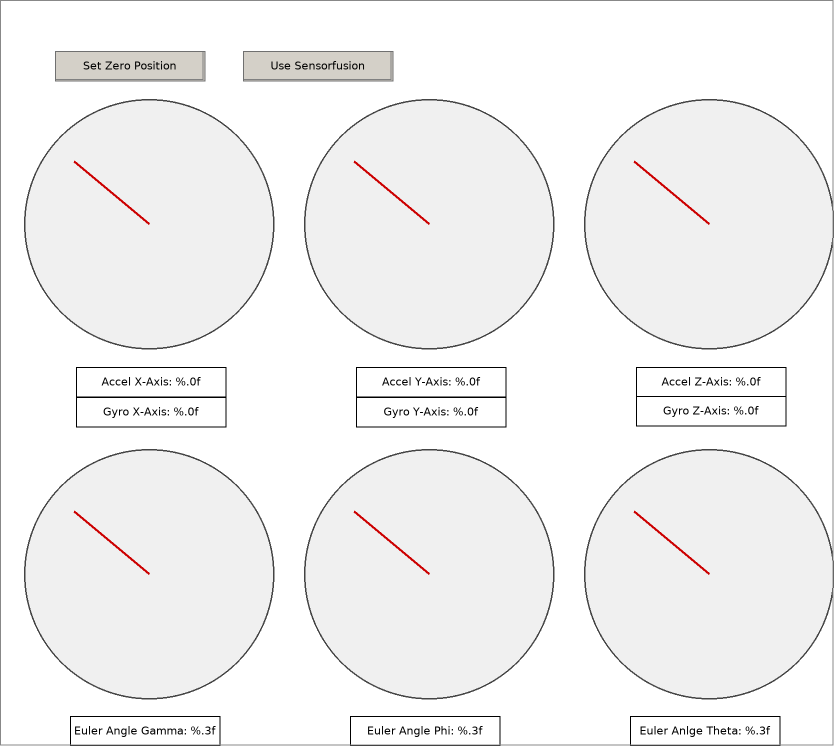
VISUALIZATION Visualization  // 834x746
    Meter360 (24,99 250x250), value: MAIN.AccAxis[0], style: Meter-Meter360-Gray, scale format: %d, scale -2000..2000
        p518627256: °
    Rectangle (76,367 150x30), "Accel X-Axis: %.0f", text variable: MAIN.AccAxis[0]
    Button (55,51 150x30), "Set Zero Position", colour toggle: MAIN.bReady
        p2175578022: 16#FF808080
        p573394764: 16#FF80FF80
        tap MAIN.bReset
    Meter360 (304,99 250x250), value: MAIN.AccAxis[1], style: Meter-Meter360-Gray, scale format: %d, scale -2000..2000
        p518627256: °
    Rectangle (356,367 150x30), "Accel Y-Axis: %.0f", text variable: MAIN.AccAxis[1]
    Meter360 (584,99 250x250), value: MAIN.AccAxis[2], style: Meter-Meter360-Gray, scale format: %d, scale -2000..2000
        p518627256: °
    Rectangle (636,367 150x30), "Accel Z-Axis: %.0f", text variable: MAIN.AccAxis[2]
    Meter360 (24,449 250x250), value: MAIN.degGamma, style: Meter-Meter360-Gray, scale format: %d, scale 0..360
        p518627256: °
    Meter360 (304,449 250x250), value: MAIN.degPhi, style: Meter-Meter360-Gray, scale format: %d, scale 0..360
        p518627256: °
    Meter360 (584,449 250x250), value: MAIN.degTheta, style: Meter-Meter360-Gray, scale format: %d, scale 0..360
        p518627256: °
    Rectangle (70,716 150x30), "Euler Angle Gamma: %.3f", text variable: MAIN.degGamma
    Rectangle (350,716 150x30), "Euler Angle Phi: %.3f", text variable: MAIN.degPhi
    Rectangle (630,716 150x30), "Euler Anlge Theta: %.3f", text variable: MAIN.degTheta
    Rectangle (76,397 150x30), "Gyro X-Axis: %.0f", text variable: MAIN.GyroAxis[0]
    Rectangle (356,397 150x30), "Gyro Y-Axis: %.0f", text variable: MAIN.GyroAxis[1]
    Rectangle (636,396 150x30), "Gyro Z-Axis: %.0f", text variable: MAIN.GyroAxis[2]
    Button (243,51 150x30), "Use Sensorfusion", colour toggle: MAIN.bUseSensorFusion
        p2175578022: 16#FF808080
        p573394764: 16#FF80FF80
        toggle MAIN.bUseSensorFusion
END_VISUALIZATION

(* stored: Version 1.1.0.1, ProductVersion 3.1.4024.13
   Visu Visualization: Id {2bcdb9c8-65b9-4a3d-9749-96111609333d} *)
